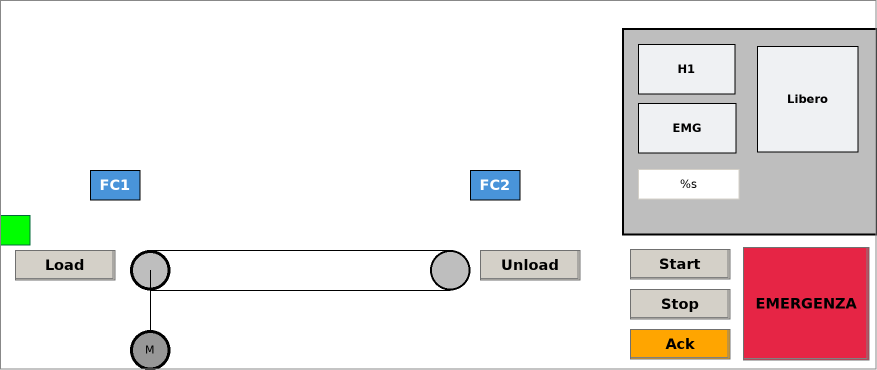
VISUALIZATION Visualization  // 877x370
    Ellipse (130,250 40x40)
    Ellipse (430,250 40x40)
    Line (150,250) (450,250)
    Line (150,290) (450,290)
    Ellipse (130,330 40x40), "M", colour toggle: GVL_IO.rawOutputs.M
    Line (150,270) (150,330)
    RoundedRectangle (622,28 255x207)
    RoundedRectangle (638,44 97x50), "H1", colour toggle: GVL_IO.rawOutputs.H1
    RoundedRectangle (638,103 98x50), "EMG", colour toggle: GVL_IO.rawOutputs.HEmg
    Textfield (638,169 101x30), "%s", text variable: MAIN.plant.simuVar.sET
    Button (630,249 100x30), "Start"
        OnMouseDown: execute { GVL_IO.rawInputs.Start := TRUE; }
        OnMouseUp: execute { GVL_IO.rawInputs.Start := FALSE; }
    Button (630,289 100x30), "Stop"
        OnMouseDown: execute { GVL_IO.rawInputs.Stop := FALSE; }
        OnMouseUp: execute { GVL_IO.rawInputs.Stop := TRUE; }
    Button (630,329 100x30), "Ack"
        OnMouseDown: execute { GVL_IO.rawInputs.Ack := TRUE; }
        OnMouseUp: execute { GVL_IO.rawInputs.Ack  := FALSE; }
    Button (743,247 126x113), "EMERGENZA"
        OnMouseDown: execute { GVL_IO.rawInputs.Emg := FALSE; }
        OnMouseUp: execute { GVL_IO.rawInputs.Emg  := TRUE; }
    RoundedRectangle (0,215 30x30), invisible if: MAIN.plant.simuVar.invis
        p3560616238: MAIN.plant.simuVar.x
    RoundedRectangle (90,170 50x30), "FC1", colour toggle: GVL_IO.rawInputs.FC1
    RoundedRectangle (470,170 50x30), "FC2", colour toggle: GVL_IO.rawInputs.FC2
    Button (15,250 100x30), "Load"
        OnMouseDown: execute { GVL_IO.rawInputs.FC1 := TRUE; }
    RoundedRectangle (757,46 101x106), "Libero", colour toggle: GVL_IO.rawOutputs.Libero
    Button (480,250 100x30), "Unload"
        OnMouseDown: execute { GVL_IO.rawInputs.FC2 := FALSE; }
END_VISUALIZATION

(* stored: Version 1.1.0.1
   Visu Visualization: Id {4c1d261f-2b67-0a03-0976-9045503e7194} *)
